# EPICS substitutions: EPICS/phoeniL300i.substitutions
file phoenixL300i.template
{
	pattern
	{ sys	sec	dev   }
	{ TEST	TEST	GLD02 }
}
